PROGRAM MAIN
VAR
END_VAR

HMI.level_1 := GVL.mb_Output_Registers[0];
HMI.level_2 := GVL.mb_Output_Registers[1];
HMI.level_3 := GVL.mb_Output_Registers[2];
HMI.pump_1 := GVL.mb_Output_Coils[0];
HMI.valve := GVL.mb_Output_Coils[1];
HMI.pump_3 := GVL.mb_Output_Coils[2];

IF HMI.level_2 >= 10 THEN
	HMI.tubeOUT_2 := TRUE;
ELSIF HMI.level_2 < 10 THEN
	HMI.tubeOUT_2 := FALSE;
END_IF;

END_PROGRAM

(* stored: Version 1.1.0.1
   POU MAIN: Id {759fd4c8-c070-42ec-8eeb-55fbb1069cba}, SpecialFunc None *)
